FUNCTION_BLOCK FB_FindAllPartProgram 
VAR_INPUT
	Execute 	: BOOL;
	sNetId		: STRING;
	sPathName	: STRING;
	StopAtEqual	: BOOL;
	NameToStop	: STRING;
END_VAR
VAR_OUTPUT
	Busy : BOOL;
	Done : BOOL;
	Error : BOOL;
	ErrorID : DINT;
	ErrorSubID : UDINT;
	filesList   : ARRAY[0..99] OF STRING;
	filesNumb	: UINT;
END_VAR
VAR
	iState : DINT := -1;
	fbEnum : FB_EnumFindFileEntry;
	RTRIG_Execute : R_TRIG;
	TON_Timeout		: TON;
	FirstChar		: STRING;
END_VAR

TON_Timeout(IN := Busy, PT := T#20S);
IF TON_Timeout.Q THEN
	fbEnum.eCmd := eEnumCmd_Abort;
	fbEnum.bExecute := TRUE;
	
	iState := 1999;
END_IF

RTRIG_Execute(CLK := Execute);
IF(RTRIG_Execute.Q) THEN
	Done := FALSE;
	Busy := TRUE;
	fbEnum.eCmd := eEnumCmd_First;
	ErrorID := 0;
	filesNumb := 0;
	MEMSET(ADR(filesList), 0, SIZEOF(filesList));
	ErrorID := 0;
	ErrorSubID := 0;
	
	iState := 0;
ELSIF NOT Execute AND NOT Busy THEN
	Busy			:= FALSE;
	Done			:= FALSE;
	Error			:= FALSE;
	
	iState := -1;
END_IF


CASE iState OF
	-1:
		;
	0:
		fbEnum.bExecute := TRUE;
		
		iState := 10;
		
	10:
		IF NOT fbEnum.bBusy THEN
            IF NOT fbEnum.bError THEN
				FirstChar := LEFT(fbEnum.stFindFile.sFileName, 1);
				IF FirstChar = 'O' THEN
					filesList[filesNumb] := fbEnum.stFindFile.sFileName;
					IF StopAtEqual AND NameToStop = filesList[filesNumb] THEN
						fbEnum.bExecute := FALSE;
					
                    	iState      := 999;
						RETURN;						
					END_IF
					filesNumb := filesNumb + 1;
				END_IF
                IF NOT fbEnum.bEOE AND filesNumb <= 99 THEN
                    fbEnum.eCmd := eEnumCmd_Next; (* enum next entry *)
					fbEnum.bExecute := FALSE;
					
                    iState      := 0;
                ELSE (* no more entries *)
					fbEnum.bExecute := FALSE;
					
                    iState      := 999;
                END_IF
            ELSE (* log error *)
				ErrorSubID := fbEnum.nErrID;
				fbEnum.bExecute := FALSE;	
			
                iState     := 1010;
            END_IF
        END_IF
		
	999:
		Busy := FALSE;
		Done := TRUE;

		
END_CASE

IF(iState > 1000) THEN
	fbEnum.bExecute := FALSE;
	Error 	:= TRUE;
	ErrorID := iState;
	Busy 	:= FALSE;
ELSE
	Error := FALSE;
END_IF

A_Call();

ACTION A_Call:
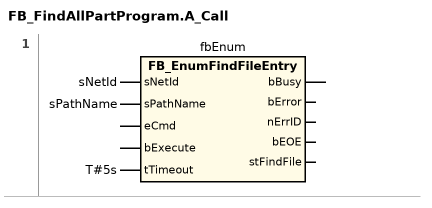
// NETWORK 1
fbEnum(sNetId := sNetId, sPathName := sPathName, tTimeout := T#5s); // FB_EnumFindFileEntry
END_ACTION

END_FUNCTION_BLOCK

(* stored: Version 1.1.0.1, ProductVersion 3.1.4024.13
   POU FB_FindAllPartProgram: Id {b08a44ff-7733-4cd1-a1dc-439b13a1af88}, SpecialFunc None
   Action A_Call: Id {b8a55894-b7b8-4454-b6cb-118f1a305209} *)
